PROGRAM _5000_PRG_Aborting
VAR_IN_OUT
    CurrentStep : ActiveStep;  // Shared step structure with state machine
END_VAR

VAR_INPUT
    StepTimerSeconds : DINT;   // Timer value from state machine
    RetrySignal : BOOL;        // Retry signal from state machine
    StateMachineStatus : ST_SM_Status;  // Complete state machine status
END_VAR

VAR_OUTPUT
    NextStep : DINT;           // Next step to transition to
END_VAR

VAR
    // Step function blocks for aborting sequence
    fbStep5000 : FB_SequenceStep;  // Abort Prepare
    fbStep5002 : FB_SequenceStep;  // Abort Execute
    
    // Step permissives (simulation for testing)
    step5000Perms : INT := -1;     // All OK for step 5000
    step5002Perms : INT := -1;     // All OK for step 5002
    
END_VAR

//=============================================================================
// PRG_Aborting - Handles ABORTING state sequence (5000-5999)
//=============================================================================
// Step numbering: 5000, 5002 (even numbers)
// Fault steps: 5001, 5003 (odd numbers, +1 of original)

//=============================================================================
// SEQUENCE CONTROL LOGIC
//=============================================================================
// Initialize sequence when first entering ABORTING state
IF StateMachineStatus.Aborting AND CurrentStep.Step = 0 THEN
    NextStep := 5000;  // Start with first aborting step
ELSE
    // Default to current step - will be overridden by active step logic below
    NextStep := CurrentStep.Step;
END_IF;

//=============================================================================
// STEP 5000 - ABORT PREPARE
//=============================================================================
fbStep5000(
    inpStep := CurrentStep.Step,
    cfgStep := 5000,
    cfgNextStep := 5002,
    inpStepTimerSeconds := StepTimerSeconds,
    inpRetry := RetrySignal,
    inpStepPermissives := step5000Perms,
    cfgStepTimeout := 5,  // 5 second timeout (quick abort)
    inpFaultStep := FALSE,
    ActiveStep := CurrentStep
);

// Step 5000 Active Logic
IF fbStep5000.outStepActive THEN
    // Permissives simulation - Simulate based on timer
    IF StepTimerSeconds < 2 THEN
        step5000Perms := 16#FFFE;  // Bit 0 not OK (not ready yet)
    ELSE
        step5000Perms := -1;  // All permissives OK
    END_IF;
    
    // HMI configuration and actions
    CurrentStep.PermsHMI.Name := 'Abort Prepare';
    CurrentStep.PermsHMI.Desc[0] := 'Emergency Stop Clear';
    CurrentStep.PermsHMI.Desc[1] := 'Safety Systems Active';
    CurrentStep.PermsHMI.Desc[2] := 'Personnel Clear';
    
    // Add any step-specific actions here
    // Example: Set emergency stop relays, activate warning lights, etc.
    
    // FB_SequenceStep determines next step automatically based on permissives
    NextStep := fbStep5000.outNextStep;
END_IF;

//=============================================================================
// STEP 5002 - ABORT EXECUTE  
//=============================================================================
fbStep5002(
    inpStep := CurrentStep.Step,
    cfgStep := 5002,
    cfgNextStep := 999,  // 0 = sequence complete
    inpStepTimerSeconds := StepTimerSeconds,
    inpRetry := RetrySignal,
    inpStepPermissives := step5002Perms,
    cfgStepTimeout := 10,  // 10 second timeout
    inpFaultStep := FALSE,
    ActiveStep := CurrentStep
);

// Step 5002 Active Logic
IF fbStep5002.outStepActive THEN
    // Permissives simulation - Simulate based on timer
    IF StepTimerSeconds < 6 THEN
        step5002Perms := 16#FFFD;  // Bit 1 not OK (abort not complete)
    ELSE
        step5002Perms := -1;  // All permissives OK
    END_IF;
    
    // HMI configuration and actions
    CurrentStep.PermsHMI.Name := 'Abort Execute';
    CurrentStep.PermsHMI.Desc[0] := 'Emergency Shutdown Active';
    CurrentStep.PermsHMI.Desc[1] := 'Systems Securing';
    CurrentStep.PermsHMI.Desc[2] := 'Safe State Reached';
    
    // Add any step-specific actions here
    // Example: Execute shutdown sequence, secure valves, stop motors, etc.
    
    // FB_SequenceStep determines next step automatically based on permissives
    NextStep := fbStep5002.outNextStep;
END_IF;

END_PROGRAM

(* stored: Version 1.1.0.1, ProductVersion 3.1.4024.13
   POU _5000_PRG_Aborting: Id {12345678-1234-1234-1234-123456789004}, SpecialFunc None *)
